TYPE SEND_CMD_DATA :
STRUCT
	DEVICE_ID       : UDINT;
	FUNCTIONCODE    : UDINT;
	STATUE          : STRING ;
END_STRUCT
END_TYPE

(* stored: Version 1.1.0.1, ProductVersion 3.1.4018.5
   DUT SEND_CMD_DATA: Id {3d2dba9e-9024-4d74-9658-c17cbe5a0389} *)
